(* IEC 61131-3 sources: ae-json-library/src, 4 files *)

(* ---- UsingDeserializer.st ---- *)
USING Simatic.Ax.Conversion;
USING AxUnit.Assert;
USING System.Strings;
USING Simatic.Ax.Json;

{TestFixture}
Class UsingDeserializer
    VAR protected
        deserializer : Deserializer;
        buffer : ARRAY[0..999] OF CHAR;

        JSON_Entry: STRING;
        key: STRING;
        len:DINT;
        keyFound: BOOL;

    END_VAR

    {Test}
    Method Public GetValue_BASIC_DATA_TYPES
        VAR
            stringValue: STRING;
            usintValue: USINT;
            intValue: INT;
        END_VAR

        //Getting JSON and convert it to ARRAY OF CHAR
        JSON_Entry := '{ "key1": "stringValue", "key2": 10, "key3": 1234, "key4": "1234"}';
        len:= Strings.ToArray(str := JSON_Entry, arr := buffer);
        //other comment
        //blabla

        //testcomment
        //Give it to the deserializer
        deserializer.SetBuffer(REF(buffer));

        //Parse string
        key:= 'key1';
        keyFound := deserializer.TryParse( key, stringValue);

        Equal(keyFound, TRUE);
        Equal(stringValue, 'stringValue');

        //Parse usint
        key:= 'key2';
        keyFound := deserializer.TryParse( key, usintValue);

        Equal(keyFound, TRUE);
        Equal(usintValue, usint#10);

        //Parse int
        key:= 'key3';
        keyFound := deserializer.TryParse( key, intValue);

        Equal(keyFound, TRUE);
        Equal(intValue, 1234);

        //FailedParsing
        key:= 'Not a key';
        keyFound := deserializer.TryParse( key, intValue);

        Equal(keyFound, FALSE);
        Equal(intValue, 0);

        //Parse foreign datatypes int to string -> possible
        key:= 'key2';
        keyFound := deserializer.TryParse( key, stringValue);

        Equal(keyFound, TRUE);
        Equal(stringValue, '10');

        //Parse foreign datatypes string to int -> possible if string is a int
        key:= 'key4';
        keyFound := deserializer.TryParse( key, intValue);

        Equal(keyFound, TRUE);
        Equal(intValue, 1234);

         //Parse foreign datatypes string to int -> False if string is not a int
         key:= 'key1';
         keyFound := deserializer.TryParse( key, intValue);

         Equal(keyFound, FALSE);
         Equal(intValue, 0);
    END_Method

    {Test}
    Method Public GetValue_ARRAY
        VAR
            stringValue: STRING;
        END_VAR

        JSON_Entry := '{ "arraykey": [1234, 5678]}';

        len:= Strings.ToArray(str := JSON_Entry, arr := buffer);
        deserializer.SetBuffer(REF(buffer));

        key:= 'arraykey';
        keyFound := deserializer.TryParse( key, stringValue);

        Equal(keyFound, TRUE);
        Equal(stringValue, '[1234, 5678]');
    END_Method

    {Test}
    Method Public GetValue_Nested
        VAR
            stringValue: STRING;
            keyArray: ARRAY[0..1] OF STRING;
        END_VAR

        JSON_Entry := '{ "key1": {"nestedkey1": "nested value", "nestedkey2": 456}}';

        len:= Strings.ToArray(str := JSON_Entry, arr := buffer);
        deserializer.SetBuffer(REF(buffer));

        //Parse string
        key:= 'key1';
        keyFound := deserializer.TryParse( key, stringValue);

        Equal(keyFound, TRUE);
        Equal(stringValue, '{"nestedkey1": "nested value", "nestedkey2": 456}'); //right now there is a 254 character limit!

        //Get Values from a nested element
        keyArray[0] := 'key1';
        keyArray[1] := 'nestedkey1';

        keyFound := deserializer.TryParse( keyArray, stringValue);

        Equal(keyFound, TRUE);
        Equal(stringValue, 'nested value');
    END_Method

    {Test}
    Method Public GetValue_Nested_in_Nested
        VAR
            stringValue: STRING;
            keyArray: ARRAY[0..2] OF STRING;
            intValue: INT;
        END_VAR

        JSON_Entry := '{ "key1": {"nestedkey1": "nested value", "nestedkey2": {"nested_nested_key" : 1234}}}';

        len:= Strings.ToArray(str := JSON_Entry, arr := buffer);
        deserializer.SetBuffer(REF(buffer));

        //Get Values from a nested element
        keyArray[0] := 'key1';
        keyArray[1] := 'nestedkey2';
        keyArray[2] := 'nested_nested_key';

        keyFound := deserializer.TryParse( keyArray, intValue);

        Equal(keyFound, TRUE);
        Equal(intValue, 1234);
    END_Method

END_CLASS

(* ---- UsingSerializer.st ---- *)
USING AxUnit.Assert;
USING System.Strings;
USING Simatic.Ax.Conversion;
USING Simatic.Ax.Json;

{TestFixture}
Class UsingSerializer
    VAR Public
        doc : JsonDocument;
        cmpBuff : ARRAY[0..20] OF CHAR;

        e : JsonBoolean := (Value := true, Key := 'test');
        b : JsonString := (Value := 'my string value', Key := 'stringKey');
    END_VAR

END_CLASS

(* ---- configuration.st ---- *)
USING Simatic.Ax.Json;
CONFIGURATION MyConfiguration
    TASK Main(Interval := T#500ms, Priority := 1);
    PROGRAM P1 WITH Main: MyProgram;

    VAR_GLOBAL
        str : STRING;
        inNanos1 : LINT;
        inNanos2 : LINT;
    END_VAR

END_CONFIGURATION

(* ---- MyProgram.st ---- *)
USING Simatic.Ax.Conversion;
USING Simatic.Ax.Json;
USING Siemens.Simatic.Clocks;

PROGRAM MyProgram
    VAR_EXTERNAL
        ActiveStep : STRING;
        SerializedDocument1 : STRING;
        TimeCreationDocument1 : LINT;
        ParsedValue1 : INT;
        SerializedDocument2 : STRING;
        TimeCreationDocument2 : LINT;
        ParsedValue2 : DINT;
    END_VAR
    VAR
        measurement : RuntimeMeasurement;
        timeOfOperations : LTIME;
        doc : JsonDocument;
        buffer : ARRAY[0..200] OF CHAR;
        cmpBuff : ARRAY[0..20] OF CHAR;
        myBoolean : JsonBoolean := (Value := TRUE, Key := 'myBoolean');
        myInt : JsonInt := (Value := 1234, Key := 'myInt');
        myDint : JsonDInt := (Value := DINT#12345678, Key := 'myDint');
        myObject : JsonObject := (Key := 'myObject');
        step : Steps;
        deserializer : Deserializer;
        keyFound : BOOL;
        keyArray : ARRAY[0..1] OF STRING := ['myObject', 'myDint'];
    END_VAR

    CASE step OF
        Steps#CreateDocument1:
            // Create Document 1st object model
            // Expected Value: {"myInt": 1234}
            ActiveStep := 'Create JSON Document {"myInt": 1234}';
            doc.AddElement(myInt);
            doc.Serialize();
            step := Steps#SerializeDocument1
            ;
        Steps#SerializeDocument1:
            // Serialize Document 1st object model1
            ActiveStep := 'Serialize JSON Document {"myInt": 1234}';
            measurement.Start();
            doc.buffer := REF(buffer);
            doc.Serialize();
            timeOfOperations := measurement.Stop();
            SerializedDocument1 := Arrays.ToString(buffer);
            TimeCreationDocument1 := measurement.GetElapsedNanoseconds();
            step := Steps#ParseDocument1
            ;
        Steps#ParseDocument1:
            // Parse Document 1st object model
            ActiveStep := 'Parse for "myInt" JSON Document {"myInt": 1234}';
            deserializer.buffer := REF(buffer);
            keyFound := deserializer.TryParse('myInt', ParsedValue1);
            step := Steps#ResetJSonDocument1
            ;
        Steps#ResetJSonDocument1:
            // ResetJSonDocument 1st object model
            ActiveStep := 'Reset JSON Document {"myInt": 1234}';
            doc.Reset();
            step := Steps#CreateDocument2
            ;
        Steps#CreateDocument2:
            // Create nested JSON document which looks like:
            // {"myBoolean": true, "myObject": {"myInt": 1234, "myDint": 12345678}}
            ActiveStep := 'Create JSON Document {"myBoolean": true, "myObject": {"myInt": 1234, "myDint": 12345678}}';
            myObject.AddElement(myInt);
            myObject.AddElement(myDint);
            doc.AddElement(myBoolean);
            doc.AddElement(myObject);
            step := Steps#SerializeDocument2
            ;
        Steps#SerializeDocument2:
            // Serialize the document {"myBoolean": true, "myObject": {"myInt": 1234, "myDint": 12345678}}
            ActiveStep := 'Serialize JSON Document {"myBoolean": true, "myObject": {"myInt": 1234, "myDint": 12345678}}';
            measurement.Start();
            doc.Serialize();
            timeOfOperations := measurement.Stop();
            SerializedDocument2 := Arrays.ToString(buffer);
            TimeCreationDocument2 := measurement.GetElapsedNanoseconds();
            step := Steps#ParseDocument2;
            ;
        Steps#ParseDocument2:
            // Parse Document for the value of the nested key `myObject.myDint` and expect `12345678`
            // Get Values from a nested element
            ActiveStep := 'Parse for "myInt" JSON Document {"myBoolean": true, "myObject": {"myInt": 1234, "myDint": 12345678}}';
            deserializer.buffer := REF(buffer);
            keyFound := deserializer.TryParse(keyArray, ParsedValue2);
            step := Steps#ResetJSonDocument2;
            ;
        Steps#ResetJSonDocument2:
            // ResetJSonDocument 2nd configuration
            ActiveStep := 'Reset JSON Document {"myBoolean": true, "myObject": {"myInt": 1234, "myDint": 12345678}}';
            doc.Reset();
            step := Steps#CreateDocument1;
            ;
    END_CASE;

END_PROGRAM

TYPE
    Steps : (
        CreateDocument1,
        SerializeDocument1,
        ParseDocument1,
        ResetJSonDocument1,
        CreateDocument2,
        SerializeDocument2,
        ParseDocument2,
        ResetJSonDocument2) := CreateDocument1;
END_TYPE
